// Mitsubishi GX Works2 project: yoavi   PLC: FX3G

// global labels: Global1
VAR_GLOBAL
  start_day AT X007 : BOOL;
  analog_output AT D8282 : INT;
  ready_packs AT D1100 : REAL;
  input_petel AT D1110 : REAL;
  input_limon AT D1120 : REAL;
  input_stable AT D1130 : REAL;
  petel_amount AT D1210 : REAL;
  stable_amount AT D1230 : REAL;
  input_bear AT D1140 : REAL;
  bear_amount AT D1240 : REAL;
  light_day AT Y007 : BOOL;
  M_10 AT M10 : BOOL;
  end_day AT X005 : BOOL;
  day_end AT X005 : BOOL;
  flavor_prepare AT X001 : BOOL;
  analog_input1 AT D8280 : INT;
  gumigam_type_input AT D7990 : REAL;
END_VAR
VAR_GLOBAL CONSTANT
  pinuk : REAL := 6;
  regular : REAL := 5;
  divide_num : REAL := 400;
END_VAR
VAR_GLOBAL
  save_analog_value AT D7990 : REAL;
  pinuk_selected AT M20 : BOOL;
  regular_selected AT M30 : BOOL;
END_VAR
VAR_GLOBAL CONSTANT
  petel_for_pinuk : REAL := 385;
END_VAR
VAR_GLOBAL
  petel_pinuk_check AT M22 : BOOL;
END_VAR
VAR_GLOBAL CONSTANT
  stable_for_pinuk : REAL := 210;
END_VAR
VAR_GLOBAL
  stable_pinuk_check AT M26 : BOOL;
END_VAR
VAR_GLOBAL CONSTANT
  bear_for_pinuk : REAL := 70;
END_VAR
VAR_GLOBAL
  bear_pinuk_check AT M28 : BOOL;
END_VAR
VAR_GLOBAL CONSTANT
  petel_for_regular : REAL := 280;
END_VAR
VAR_GLOBAL
  petel_regular_check AT M32 : BOOL;
END_VAR
VAR_GLOBAL CONSTANT
  stable_for_regular : REAL := 105;
END_VAR
VAR_GLOBAL
  stable_regular_check AT M36 : BOOL;
  bear_regular_check AT M38 : BOOL;
END_VAR
VAR_GLOBAL CONSTANT
  bear_for_regular : REAL := 28;
END_VAR
VAR_GLOBAL
  limon_pinuk_check AT M24 : BOOL;
END_VAR
VAR_GLOBAL CONSTANT
  limon_for_pinuk : REAL := 665;
END_VAR
VAR_GLOBAL
  pinuk_available AT M120 : BOOL;
END_VAR
VAR_GLOBAL CONSTANT
  limon_for_regular : REAL := 455;
END_VAR
VAR_GLOBAL
  limon_regular_check AT M34 : BOOL;
  limon_amount AT D1220 : REAL;
  regular_available AT M130 : BOOL;
  start_cooking AT X001 : BOOL;
  make_ice_cream AT X001 : BOOL;
  shortage AT M10 : BOOL;
END_VAR
VAR_GLOBAL CONSTANT
  petel_for_petel_regular : REAL := 280;
END_VAR
VAR_GLOBAL
  petel_basket AT D1310 : REAL;
END_VAR
VAR_GLOBAL CONSTANT
  limon_for_petel_regular : REAL := 35;
  stable_for_petel_regular : REAL := 35;
  petel_for_limon_regular : REAL;
END_VAR
VAR_GLOBAL
  limon_basket AT D1320 : REAL;
END_VAR
VAR_GLOBAL CONSTANT
  limon_for_limon_regular : REAL := 420;
  stable_for_limon_regular : REAL := 70;
  petel_for_petel_pinuk : REAL := 385;
  limon_for_petel_pinuk : REAL := 105;
  stable_for_petel_pinuk : REAL := 70;
  petel_for_limon_pinuk : REAL;
  limon_for_limon_pinuk : REAL := 560;
  stable_for_limon_pinuk : REAL := 140;
  petel_ingredients_regular : REAL := 364;
  limon_ingredients_regular : REAL := 504;
  petel_ingredients_pinuk : REAL := 595;
  limon_ingredients_pinuk : REAL := 735;
END_VAR
VAR_GLOBAL
  tc1 AT TC1 : BOOL;
  check_light AT TS1 : BOOL;
  prepare_light AT Y000 : BOOL;
END_VAR
VAR_GLOBAL CONSTANT
  timer_preparing : INT := 50;
END_VAR
VAR_GLOBAL
  start_freezing AT X002 : BOOL;
  ready_to_freez AT M42 : BOOL;
  petel_basket_cold AT D1410 : REAL;
  limon_basket_cold AT D1420 : REAL;
  tc2 AT TC2 : BOOL;
END_VAR
VAR_GLOBAL CONSTANT
  timer_freezing : INT := 80;
END_VAR
VAR_GLOBAL
  freezing_light AT Y002 : BOOL;
  check_light2 AT TS2 : BOOL;
  temprature_sens AT X003 : BOOL;
  ready_to_mix AT M44 : BOOL;
  tc_4 AT TC4 : BOOL;
  tc_3 AT TC3 : BOOL;
END_VAR
VAR_GLOBAL CONSTANT
  regular_mix_time : INT := 30;
  pinuk_mix_time : INT := 50;
END_VAR
VAR_GLOBAL
  tc_5 AT TC5 : BOOL;
  tc_6 AT TC6 : BOOL;
  y_5 AT Y005 : BOOL;
  y_6 AT Y006 : BOOL;
END_VAR
VAR_GLOBAL CONSTANT
  blink_time : INT := 5;
END_VAR
VAR_GLOBAL
  M_0 AT M0 : BOOL;
  ts_5 AT TS5 : BOOL;
  ts_6 AT TS6 : BOOL;
  M_1 AT M1 : BOOL;
  limon_mix_basket AT D1520 : REAL;
  petel_mix_basket AT D1510 : REAL;
  start_packing AT X004 : BOOL;
  M_16 AT M16 : BOOL;
  one_unit_start AT CC1 : BOOL;
END_VAR
VAR_GLOBAL CONSTANT
  one_unit_packed : REAL := 1;
  first_unit_packed : REAL := 5;
  first_start : REAL := 5;
END_VAR
VAR_GLOBAL
  full_pack AT CC2 : BOOL;
  one_unit_packing AT X000 : BOOL;
  first_in_pack AT CS1 : BOOL;
  last_in_pack AT CS2 : BOOL;
END_VAR
VAR_GLOBAL CONSTANT
  seven_units : REAL := 7;
  pack_full : REAL := 7;
END_VAR
VAR_GLOBAL
  packing_in_process AT Y004 : BOOL;
  packing_end AT M11 : BOOL;
  ts_3 AT TS3 : BOOL;
  ts_4 AT TS4 : BOOL;
  reset_counters AT X001 : BOOL;
END_VAR
VAR_GLOBAL CONSTANT
  add_1 : REAL := 1;
END_VAR
VAR_GLOBAL
  analog_light AT M50 : BOOL;
END_VAR
VAR_GLOBAL CONSTANT
  Mul_num : INT := 400;
  one_gumigum : INT := 1;
  one_icecream : REAL := 6;
  one_ice_cream : REAL := 5;
  seven_icecream : REAL := 7;
END_VAR
VAR_GLOBAL
  cc1 AT CC1 : BOOL;
  cc2 AT CC2 : BOOL;
END_VAR
VAR_GLOBAL CONSTANT
  seven_gumigum : INT := 7;
END_VAR
VAR_GLOBAL
  first_gumigum AT M13 : BOOL;
  cs1 AT CS1 : BOOL;
END_VAR

// task Task_01 (event TRUE, interval 0, priority 31): POU_01

PROGRAM POU_01
(* structured ladder/FBD written out as ST: instructions are called as NAME(EN, inputs, outputs); _pN, _eN, _tN stand for wires *)
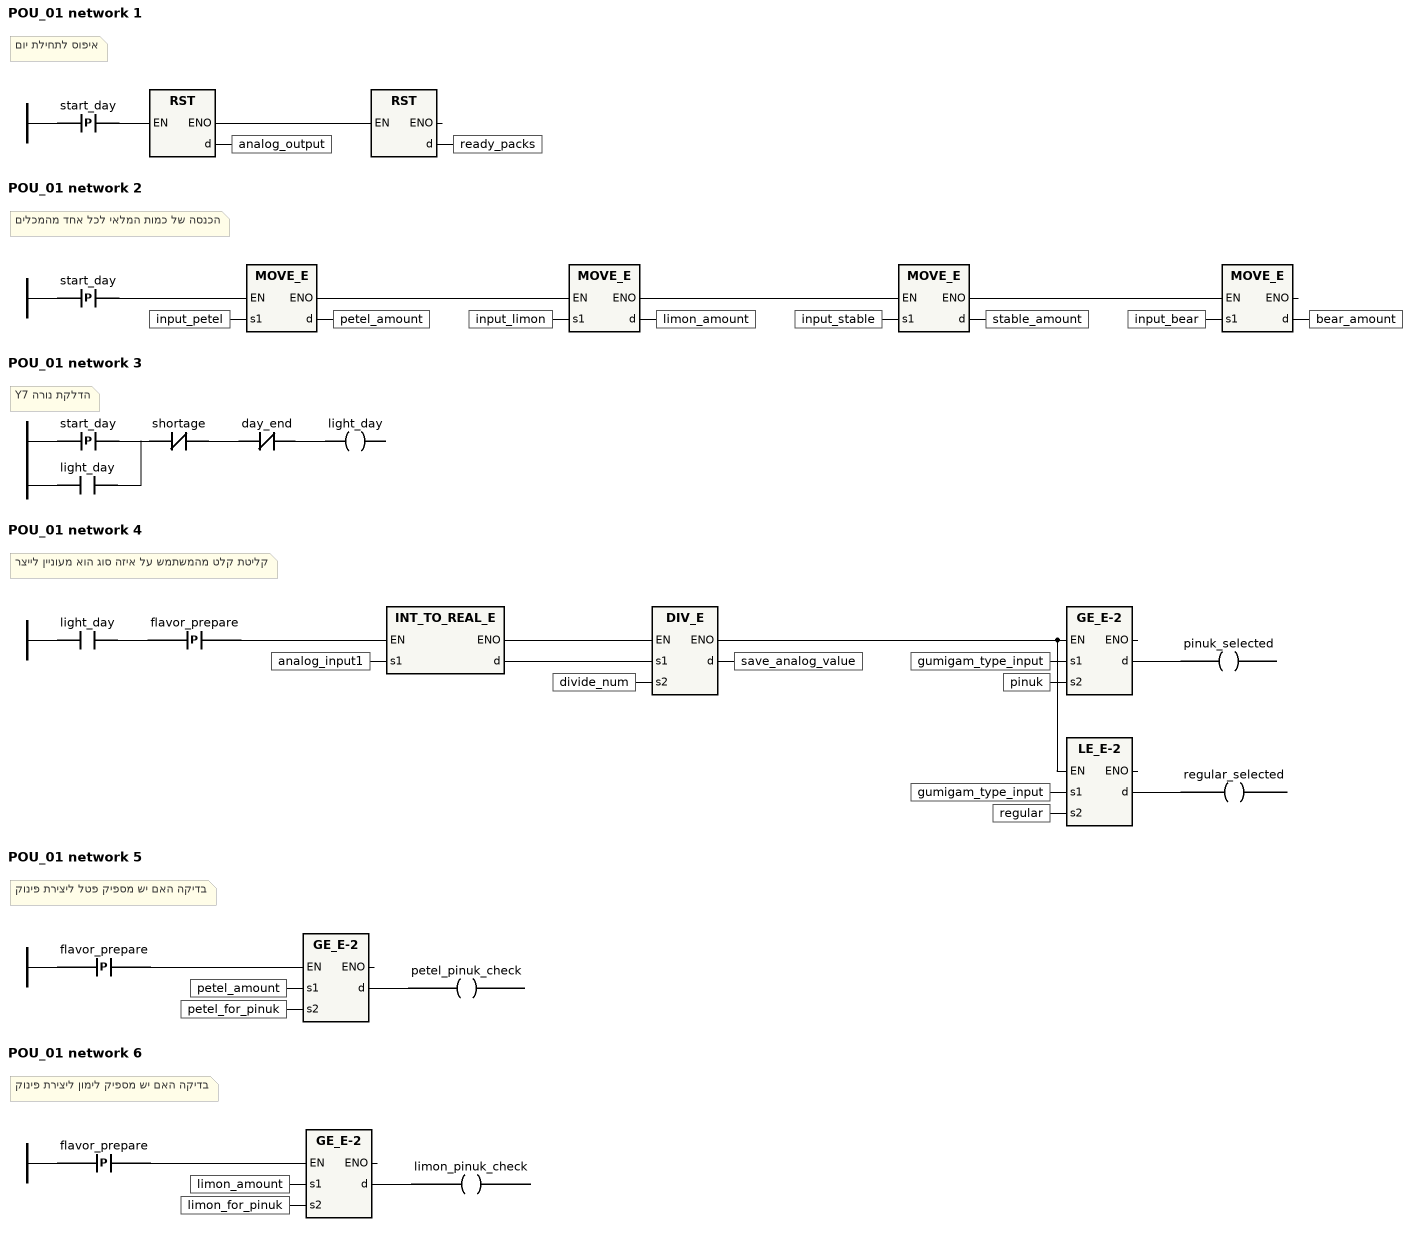
(* network 1 *)
(* איפוס לתחילת יום *)
_e1 := RST(LDP(TRUE, start_day), analog_output);
RST(_e1, ready_packs);
(* network 2 *)
(* הכנסה של כמות המלאי לכל אחד מהמכלים *)
_e1 := MOVE_E(LDP(TRUE, start_day), input_petel, petel_amount);
_e2 := MOVE_E(_e1, input_limon, limon_amount);
_e3 := MOVE_E(_e2, input_stable, stable_amount);
MOVE_E(_e3, input_bear, bear_amount);
(* network 3 *)
(* הדלקת נורה Y7 *)
light_day := ((LDP(TRUE, start_day) OR light_day) AND NOT shortage) AND NOT day_end;
(* network 4 *)
(* קליטת קלט מהמשתמש על איזה סוג הוא מעוניין לייצר *)
_e2 := INT_TO_REAL_E(light_day AND LDP(TRUE, flavor_prepare), analog_input1, _t1);
_e3 := DIV_E(_e2, _t1, divide_num, save_analog_value);
GE_E(_e3, gumigam_type_input, pinuk, _t4);
pinuk_selected := _t4;
LE_E(_e3, gumigam_type_input, regular, _t5);
regular_selected := _t5;
(* network 5 *)
(* בדיקה האם יש מספיק פטל ליצירת פינוק *)
GE_E(LDP(TRUE, flavor_prepare), petel_amount, petel_for_pinuk, _t1);
petel_pinuk_check := _t1;
(* network 6 *)
(* בדיקה האם יש מספיק לימון ליצירת פינוק *)
GE_E(LDP(TRUE, flavor_prepare), limon_amount, limon_for_pinuk, _t1);
limon_pinuk_check := _t1;
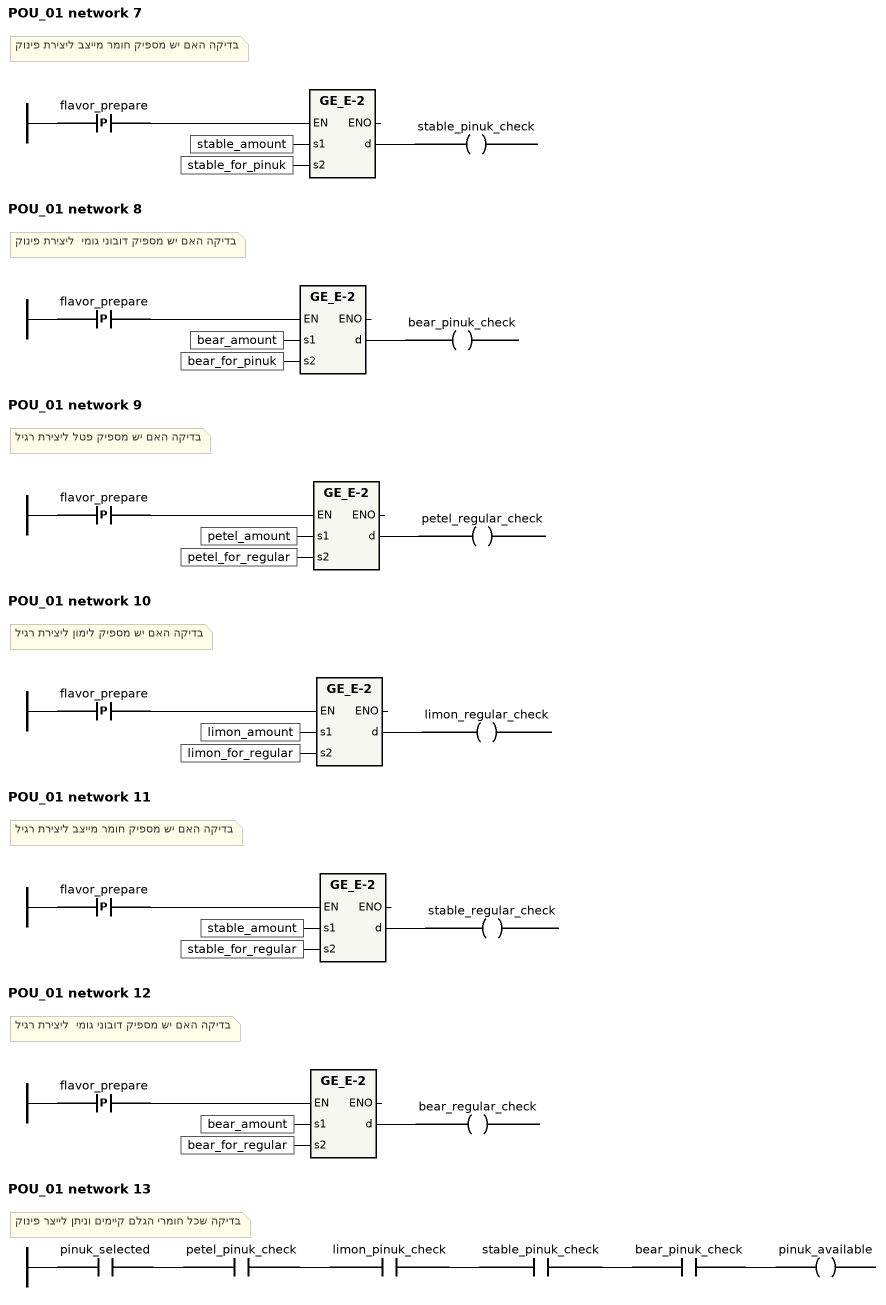
(* network 7 *)
(* בדיקה האם יש מספיק חומר מייצב ליצירת פינוק *)
GE_E(LDP(TRUE, flavor_prepare), stable_amount, stable_for_pinuk, _t1);
stable_pinuk_check := _t1;
(* network 8 *)
(* בדיקה האם יש מספיק דובוני גומי  ליצירת פינוק *)
GE_E(LDP(TRUE, flavor_prepare), bear_amount, bear_for_pinuk, _t1);
bear_pinuk_check := _t1;
(* network 9 *)
(* בדיקה האם יש מספיק פטל ליצירת רגיל *)
GE_E(LDP(TRUE, flavor_prepare), petel_amount, petel_for_regular, _t1);
petel_regular_check := _t1;
(* network 10 *)
(* בדיקה האם יש מספיק לימון ליצירת רגיל *)
GE_E(LDP(TRUE, flavor_prepare), limon_amount, limon_for_regular, _t1);
limon_regular_check := _t1;
(* network 11 *)
(* בדיקה האם יש מספיק חומר מייצב ליצירת רגיל *)
GE_E(LDP(TRUE, flavor_prepare), stable_amount, stable_for_regular, _t1);
stable_regular_check := _t1;
(* network 12 *)
(* בדיקה האם יש מספיק דובוני גומי  ליצירת רגיל *)
GE_E(LDP(TRUE, flavor_prepare), bear_amount, bear_for_regular, _t1);
bear_regular_check := _t1;
(* network 13 *)
(* בדיקה שכל חומרי הגלם קיימים וניתן לייצר פינוק *)
pinuk_available := pinuk_selected AND petel_pinuk_check AND limon_pinuk_check AND stable_pinuk_check AND bear_pinuk_check;
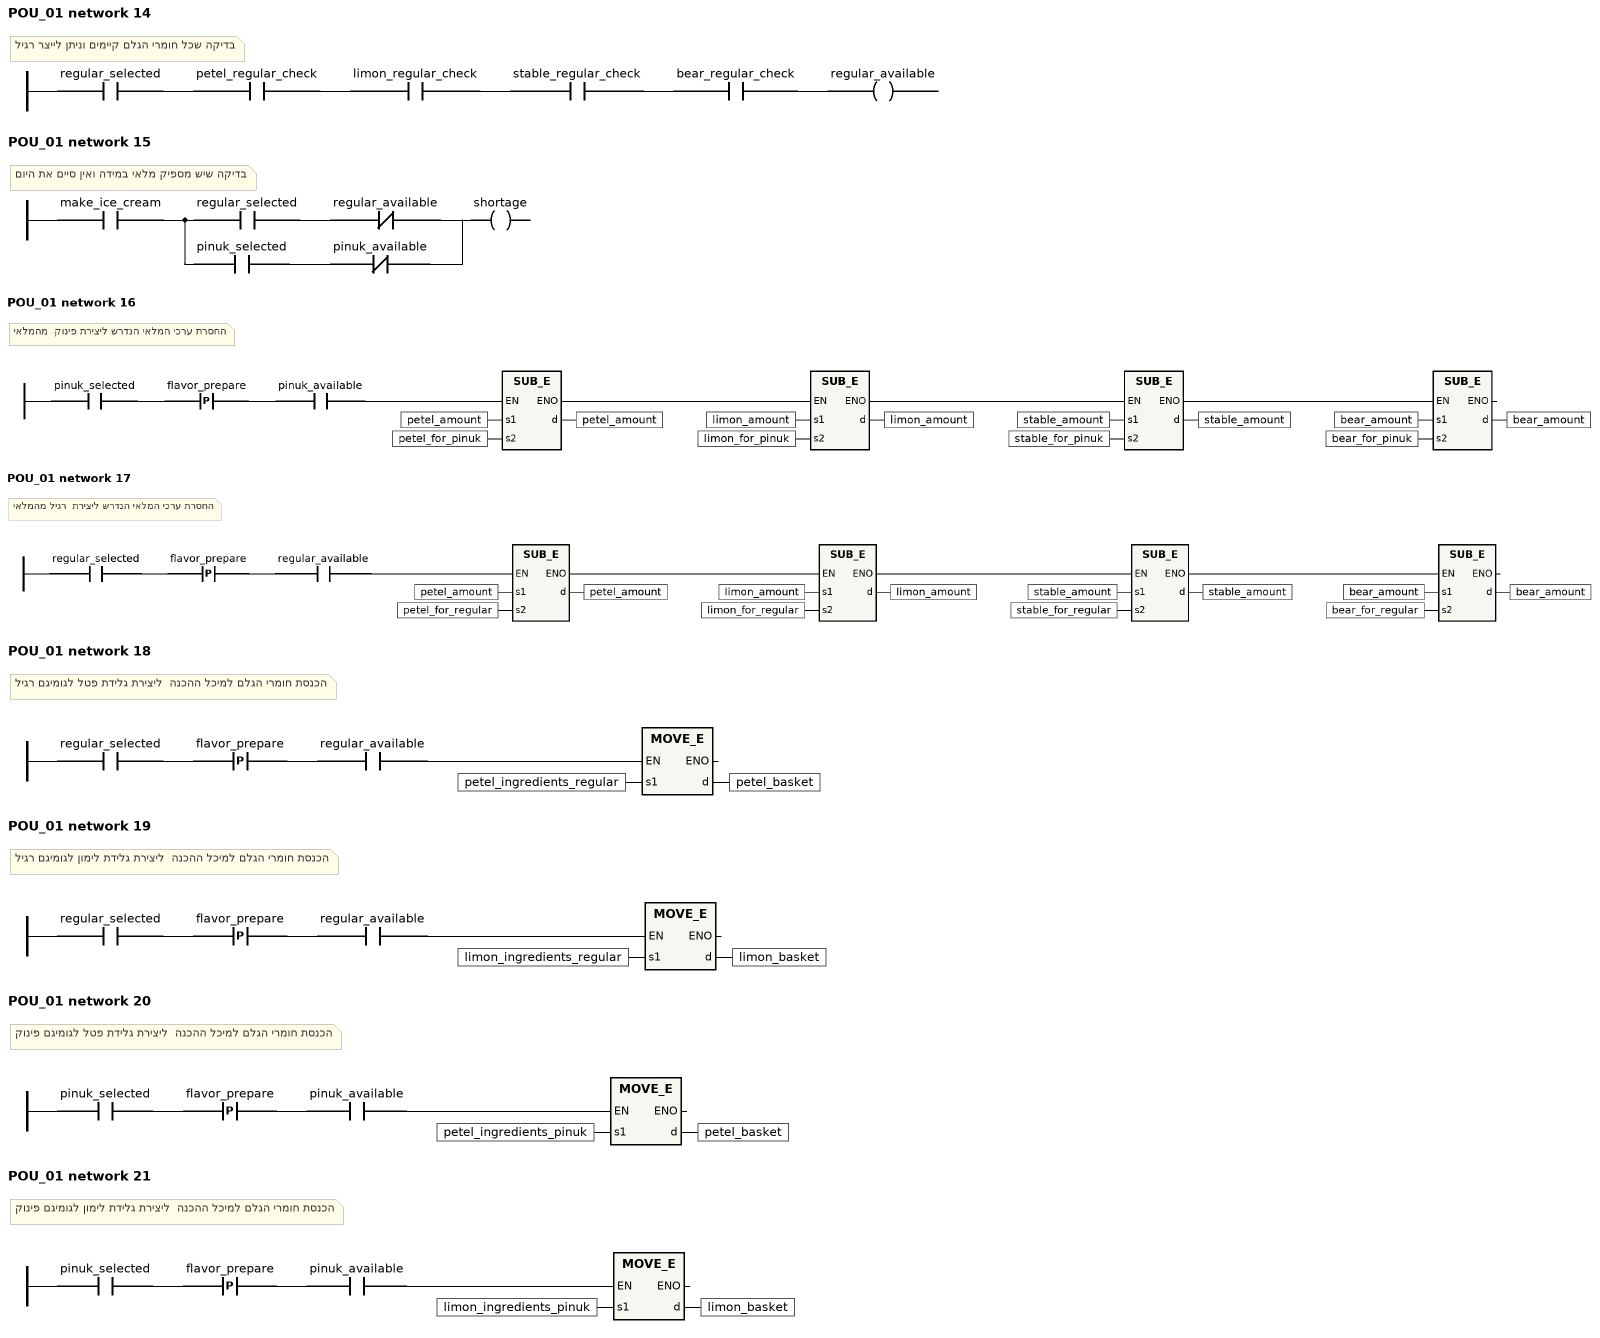
(* network 14 *)
(* בדיקה שכל חומרי הגלם קיימים וניתן לייצר רגיל *)
regular_available := regular_selected AND petel_regular_check AND limon_regular_check AND stable_regular_check AND bear_regular_check;
(* network 15 *)
(* בדיקה שיש מספיק מלאי במידה ואין סיים את היום *)
shortage := (make_ice_cream AND regular_selected AND NOT regular_available) OR (make_ice_cream AND pinuk_selected AND NOT pinuk_available);
(* network 16 *)
(* החסרת ערכי המלאי הנדרש ליצירת פינוק  מהמלאי *)
_e1 := SUB_E(pinuk_selected AND LDP(TRUE, flavor_prepare) AND pinuk_available, petel_amount, petel_for_pinuk, petel_amount);
_e2 := SUB_E(_e1, limon_amount, limon_for_pinuk, limon_amount);
_e3 := SUB_E(_e2, stable_amount, stable_for_pinuk, stable_amount);
SUB_E(_e3, bear_amount, bear_for_pinuk, bear_amount);
(* network 17 *)
(* החסרת ערכי המלאי הנדרש ליצירת  רגיל מהמלאי *)
_e1 := SUB_E(regular_selected AND LDP(TRUE, flavor_prepare) AND regular_available, petel_amount, petel_for_regular, petel_amount);
_e2 := SUB_E(_e1, limon_amount, limon_for_regular, limon_amount);
_e3 := SUB_E(_e2, stable_amount, stable_for_regular, stable_amount);
SUB_E(_e3, bear_amount, bear_for_regular, bear_amount);
(* network 18 *)
(* הכנסת חומרי הגלם למיכל ההכנה  ליצירת גלידת פטל לגומיגם רגיל *)
MOVE_E(regular_selected AND LDP(TRUE, flavor_prepare) AND regular_available, petel_ingredients_regular, petel_basket);
(* network 19 *)
(* הכנסת חומרי הגלם למיכל ההכנה  ליצירת גלידת לימון לגומיגם רגיל *)
MOVE_E(regular_selected AND LDP(TRUE, flavor_prepare) AND regular_available, limon_ingredients_regular, limon_basket);
(* network 20 *)
(* הכנסת חומרי הגלם למיכל ההכנה  ליצירת גלידת פטל לגומיגם פינוק *)
MOVE_E(pinuk_selected AND LDP(TRUE, flavor_prepare) AND pinuk_available, petel_ingredients_pinuk, petel_basket);
(* network 21 *)
(* הכנסת חומרי הגלם למיכל ההכנה  ליצירת גלידת לימון לגומיגם פינוק *)
MOVE_E(pinuk_selected AND LDP(TRUE, flavor_prepare) AND pinuk_available, limon_ingredients_pinuk, limon_basket);
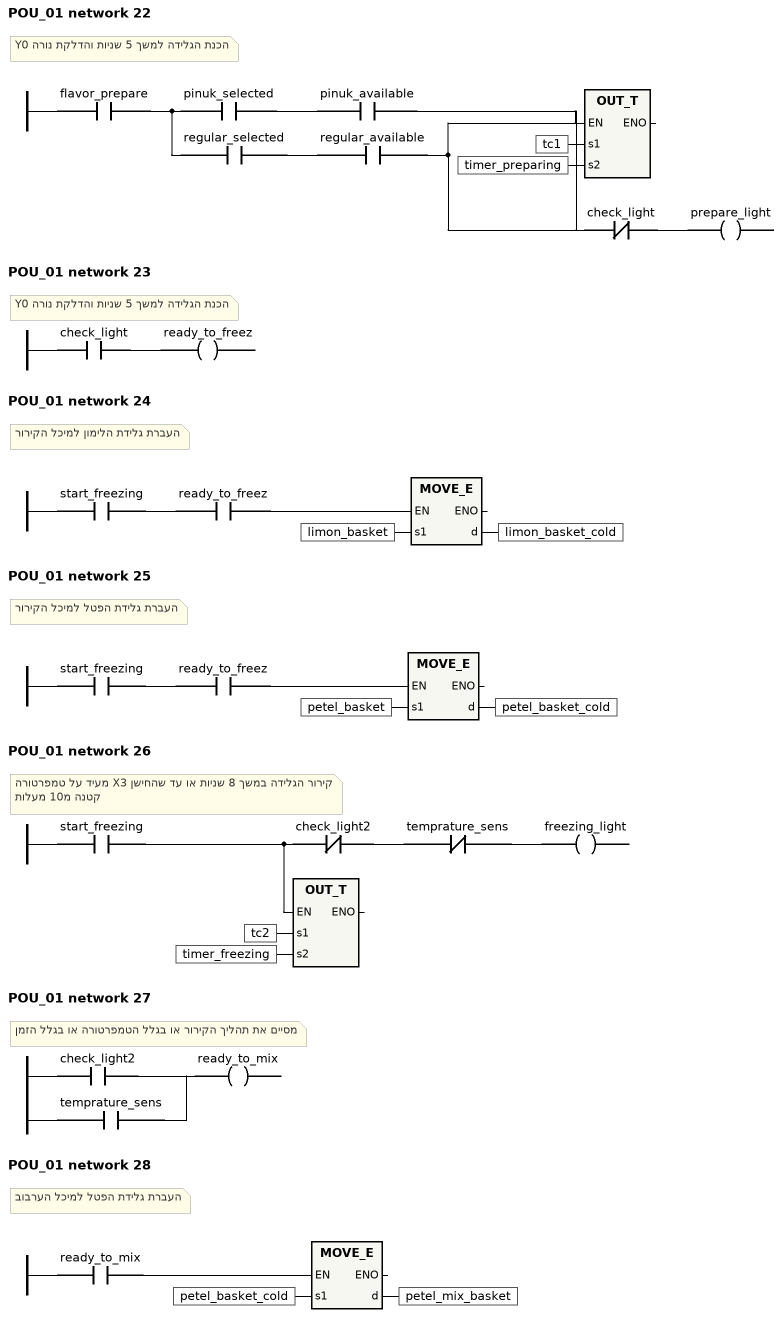
(* network 22 *)
(* הכנת הגלידה למשך 5 שניות והדלקת נורה Y0 *)
_p1 := (flavor_prepare AND pinuk_selected AND pinuk_available) OR (flavor_prepare AND regular_selected AND regular_available);
prepare_light := _p1 AND NOT check_light;
OUT_T(_p1, tc1, timer_preparing);
(* network 23 *)
(* הכנת הגלידה למשך 5 שניות והדלקת נורה Y0 *)
ready_to_freez := check_light;
(* network 24 *)
(* העברת גלידת הלימון למיכל הקירור *)
MOVE_E(start_freezing AND ready_to_freez, limon_basket, limon_basket_cold);
(* network 25 *)
(* העברת גלידת הפטל למיכל הקירור *)
MOVE_E(start_freezing AND ready_to_freez, petel_basket, petel_basket_cold);
(* network 26 *)
(* קירור הגלידה במשך 8 שניות או עד שהחישן X3 מעיד על טמפרטורה קטנה מ10 מעלות *)
freezing_light := start_freezing AND NOT check_light2 AND NOT temprature_sens;
OUT_T(start_freezing, tc2, timer_freezing);
(* network 27 *)
(* מסיים את תהליך הקירור או בגלל הטמפרטורה או בגלל הזמן *)
ready_to_mix := check_light2 OR temprature_sens;
(* network 28 *)
(* העברת גלידת הפטל למיכל הערבוב *)
MOVE_E(ready_to_mix, petel_basket_cold, petel_mix_basket);
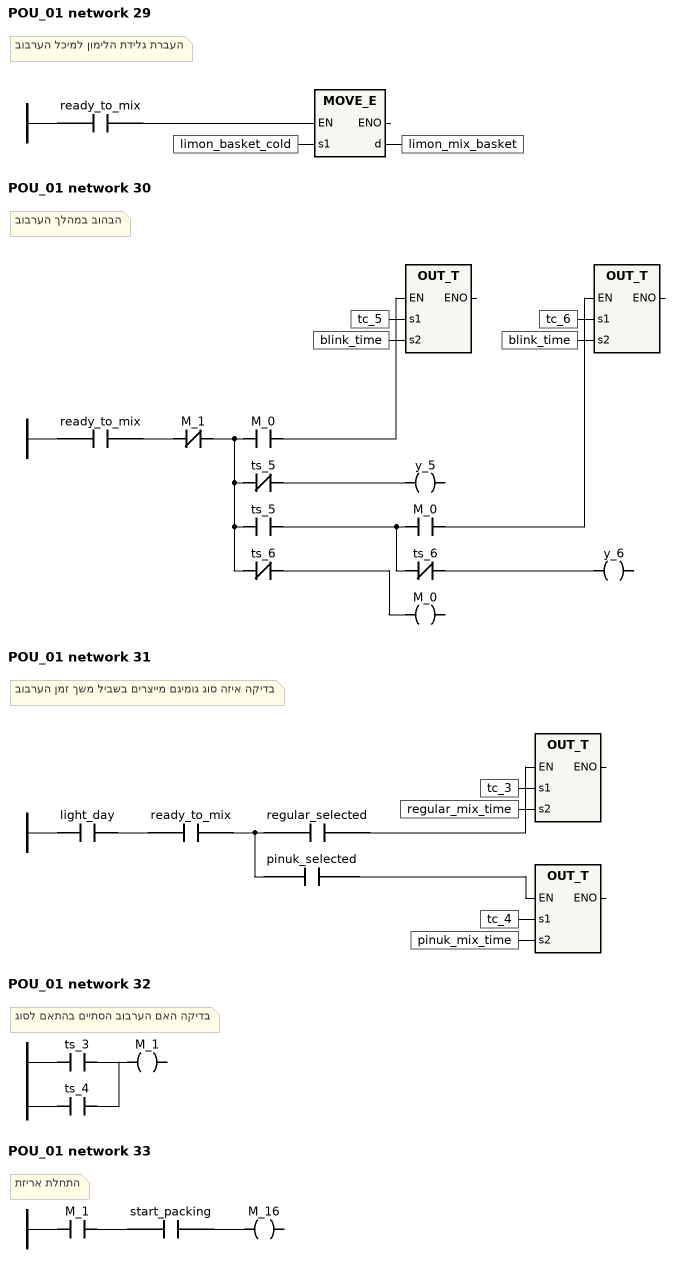
(* network 29 *)
(* העברת גלידת הלימון למיכל הערבוב *)
MOVE_E(ready_to_mix, limon_basket_cold, limon_mix_basket);
(* network 30 *)
(* הבהוב במהלך הערבוב *)
_p1 := ready_to_mix AND NOT M_1;
OUT_T(_p1 AND M_0, tc_5, blink_time);
y_5 := _p1 AND NOT ts_5;
_p2 := _p1 AND ts_5;
OUT_T(_p2 AND M_0, tc_6, blink_time);
y_6 := _p2 AND NOT ts_6;
M_0 := _p1 AND NOT ts_6;
(* network 31 *)
(* בדיקה איזה סוג גומיגם מייצרים בשביל משך זמן הערבוב *)
_p1 := light_day AND ready_to_mix;
OUT_T(_p1 AND regular_selected, tc_3, regular_mix_time);
OUT_T(_p1 AND pinuk_selected, tc_4, pinuk_mix_time);
(* network 32 *)
(* בדיקה האם הערבוב הסתיים בהתאם לסוג *)
M_1 := ts_3 OR ts_4;
(* network 33 *)
(* התחלת אריזת *)
M_16 := M_1 AND start_packing;
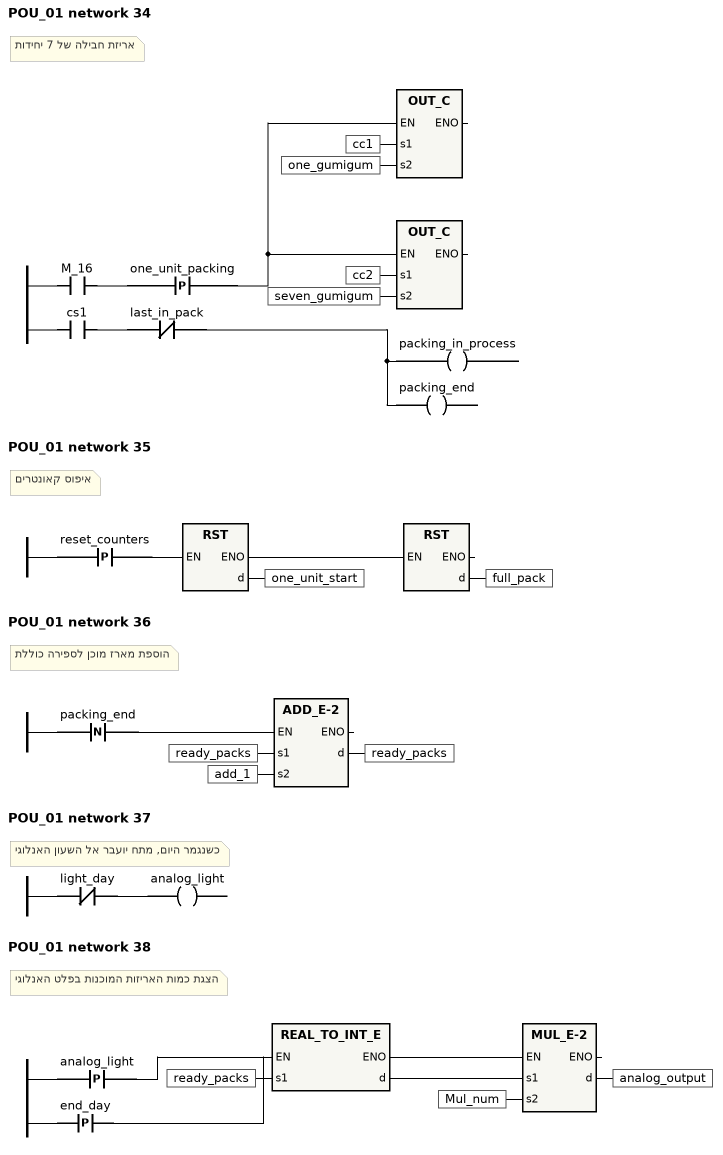
(* network 34 *)
(* אריזת חבילה של 7 יחידות *)
_p1 := M_16 AND LDP(TRUE, one_unit_packing);
OUT_C(_p1, cc1, one_gumigum);
OUT_C(_p1, cc2, seven_gumigum);
_p2 := cs1 AND NOT last_in_pack;
packing_in_process := _p2;
packing_end := _p2;
(* network 35 *)
(* איפוס קאונטרים *)
_e1 := RST(LDP(TRUE, reset_counters), one_unit_start);
RST(_e1, full_pack);
(* network 36 *)
(* הוספת מארז מוכן לספירה כוללת *)
ADD_E(LDF(TRUE, packing_end), ready_packs, add_1, ready_packs);
(* network 37 *)
(* כשנגמר היום, מתח יועבר אל השעון האנלוגי *)
analog_light := NOT light_day;
(* network 38 *)
(* הצגת כמות האריזות המוכנות בפלט האנלוגי *)
_e2 := REAL_TO_INT_E(LDP(TRUE, analog_light) OR LDP(TRUE, end_day), ready_packs, _t1);
MUL_E(_e2, _t1, Mul_num, analog_output);
END_PROGRAM
